FUNCTION_BLOCK SEL_ARRAY (* See SEL_ANY *)
  (* Standard: 61131-3 *)
  (* Version 0.0, 2004-12-15, JHC, Rockwell Automation, Converted from SRC format. *)
  (* Compiler header: package fb.rt.plc.select; *)
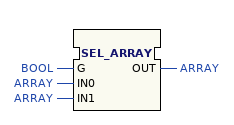
  VAR_INPUT
    G : BOOL;
    IN0 : ARRAY;
    IN1 : ARRAY;
  END_VAR
  VAR_OUTPUT
    OUT : ARRAY;
  END_VAR
END_FUNCTION_BLOCK
